	30:
		bBusy := TRUE;
		bPredictionPending := TRUE;
		IF fbMlSvr.Predict(
			pDataIn := ADR(stModelInput),
			nDataInSize := SIZEOF(ST_Wave41SmoothL1RobustLossInput),
			pDataOut := ADR(stModelOutput),
			nDataOutSize := SIZEOF(ST_Wave41SmoothL1RobustLossOutput),
			nTimeout := nPredictTimeout,
			nPriority := nPriority) THEN
			nErrorCode := fbMlSvr.nErrorCode;
			bError := fbMlSvr.bError OR (nErrorCode <> 0);
			nMaxInferenceDuration := fbMlSvr.nMaxInferenceDuration;
			bPredictionPending := FALSE;
			bBusy := FALSE;
			IF NOT(bError) THEN
				aPredictionOutput[0] := stModelOutput.out_prediction_tensor[0,0];
				FOR nOutputIndex := 1 TO 8 DO
					aPredictionOutput[nOutputIndex] := 0.0;
				END_FOR
				bPredictionReady := TRUE;
				nState := 20;
			ELSE
				nState := 90;
			END_IF
		END_IF

	90:
		bBusy := FALSE;
		bPredictionPending := FALSE;
		bError := TRUE;
END_CASE

nErrorCode := fbMlSvr.nErrorCode;
nMaxInferenceDuration := fbMlSvr.nMaxInferenceDuration;

END_FUNCTION_BLOCK

// ---- POUs/FB_Wave42GaussianNllTf3820Runner.TcPOU
FUNCTION_BLOCK FB_Wave42GaussianNllTf3820Runner
VAR_INPUT
	sModelJsonFilePath	: T_MaxString;
	sMlSvrNetId			: T_MaxString := 'local';
	eExecutionProvider	: E_ExecutionProvider := E_ExecutionProvider.CPU;
	bEnable				: BOOL;
	bReset					: BOOL;
	bLoadModel			: BOOL;
	nConfigureTimeout	: UDINT := 1000;
	nPredictTimeout		: UDINT := 100;
	nPriority			: UDINT := 0;
	fTheta					: REAL;
	fThetaDot				: REAL;
	fTorque				: REAL;
	fTemperature			: REAL;
	fDirectionFlag		: REAL;
	fThetaStep			: REAL := 0.25;
END_VAR
VAR
	fbMlSvr				: FB_MlSvrPrediction;
	stModelInput		: ST_Wave42GaussianNllInput;
	stModelOutput		: ST_Wave42GaussianNllOutput;
	rtrig_model			: R_TRIG;
	nState					: INT := 0;
	nSequenceIndex		: INT;
	nOutputIndex		: INT;
END_VAR
VAR_OUTPUT
	bConfigured			: BOOL;
	bBusy					: BOOL;
	bPredictionPending	: BOOL;
	bPredictionReady	: BOOL;
	bResetDone			: BOOL;
	bError					: BOOL;
	nErrorCode			: HRESULT;
	nMaxInferenceDuration	: UDINT;
	aPredictionOutput	: ARRAY[0..8] OF REAL;
END_VAR

rtrig_model(CLK := bLoadModel);

IF rtrig_model.Q THEN
	bPredictionPending := FALSE;
	bPredictionReady := FALSE;
	bResetDone := FALSE;
	bError := FALSE;
	IF fbMlSvr.bConfigured THEN
		nState := 5;
	ELSE
		bConfigured := FALSE;
		nState := 10;
	END_IF
END_IF

IF bReset THEN
	bPredictionPending := FALSE;
	bPredictionReady := FALSE;
	bError := FALSE;
	IF fbMlSvr.bConfigured THEN
		nState := 5;
	ELSE
		bConfigured := FALSE;
		bResetDone := TRUE;
		nState := 0;
	END_IF
END_IF

CASE nState OF
	0:
		bBusy := FALSE;
		IF bLoadModel AND NOT(bConfigured) AND NOT(bReset) THEN
			nState := 10;
		END_IF

	5:
		bBusy := TRUE;
		IF fbMlSvr.Deconfigure(nTimeout := nConfigureTimeout) THEN
			nErrorCode := fbMlSvr.nErrorCode;
			bError := fbMlSvr.bError OR (nErrorCode <> 0);
			bConfigured := FALSE;
			bBusy := FALSE;
			bResetDone := NOT(bError);
			IF bError THEN
				nState := 90;
			ELSIF bReset THEN
				nState := 0;
			ELSE
				nState := 10;
			END_IF
		END_IF

	10:
		bBusy := TRUE;
		fbMlSvr.stPredictionParameter.sMlModelFilePath := sModelJsonFilePath;
		fbMlSvr.stPredictionParameter.sMlSvrNetId := sMlSvrNetId;
		fbMlSvr.stPredictionParameter.eExecutionProvider := eExecutionProvider;
		IF fbMlSvr.Configure(nTimeout := nConfigureTimeout, nPriority := nPriority) THEN
			nErrorCode := fbMlSvr.nErrorCode;
			bError := fbMlSvr.bError OR (nErrorCode <> 0);
			bConfigured := fbMlSvr.bConfigured AND NOT(bError);
			bBusy := FALSE;
			IF bConfigured THEN
				nState := 20;
			ELSE
				nState := 90;
			END_IF
		END_IF

	20:
		bBusy := FALSE;
		bPredictionPending := FALSE;
		IF bEnable AND bConfigured AND NOT(bError) AND NOT(bReset) THEN
			FOR nSequenceIndex := 0 TO 32 DO
				stModelInput.in_input_tensor[0,nSequenceIndex,0] := fTheta + (INT_TO_REAL(nSequenceIndex) * fThetaStep);
				stModelInput.in_input_tensor[0,nSequenceIndex,1] := fThetaDot;
				stModelInput.in_input_tensor[0,nSequenceIndex,2] := fTorque;
				stModelInput.in_input_tensor[0,nSequenceIndex,3] := fTemperature;
			END_FOR
			bPredictionReady := FALSE;
			bPredictionPending := TRUE;
			nState := 30;
		END_IF

	30:
		bBusy := TRUE;
		bPredictionPending := TRUE;
		IF fbMlSvr.Predict(
			pDataIn := ADR(stModelInput),
			nDataInSize := SIZEOF(ST_Wave42GaussianNllInput),
			pDataOut := ADR(stModelOutput),
			nDataOutSize := SIZEOF(ST_Wave42GaussianNllOutput),
			nTimeout := nPredictTimeout,
			nPriority := nPriority) THEN
			nErrorCode := fbMlSvr.nErrorCode;
			bError := fbMlSvr.bError OR (nErrorCode <> 0);
			nMaxInferenceDuration := fbMlSvr.nMaxInferenceDuration;
			bPredictionPending := FALSE;
			bBusy := FALSE;
			IF NOT(bError) THEN
				aPredictionOutput[0] := stModelOutput.out_prediction_tensor[0,0];
				aPredictionOutput[1] := stModelOutput.out_prediction_tensor[0,1];
				FOR nOutputIndex := 2 TO 8 DO
					aPredictionOutput[nOutputIndex] := 0.0;
				END_FOR
				bPredictionReady := TRUE;
				nState := 20;
			ELSE
				nState := 90;
			END_IF
		END_IF

	90:
		bBusy := FALSE;
		bPredictionPending := FALSE;
		bError := TRUE;
END_CASE

nErrorCode := fbMlSvr.nErrorCode;
nMaxInferenceDuration := fbMlSvr.nMaxInferenceDuration;

END_FUNCTION_BLOCK

// ---- POUs/FB_Wave42QuantileP10P50P90Tf3820Runner.TcPOU
FUNCTION_BLOCK FB_Wave42QuantileP10P50P90Tf3820Runner
VAR_INPUT
	sModelJsonFilePath	: T_MaxString;
	sMlSvrNetId			: T_MaxString := 'local';
	eExecutionProvider	: E_ExecutionProvider := E_ExecutionProvider.CPU;
	bEnable				: BOOL;
	bReset					: BOOL;
	bLoadModel			: BOOL;
	nConfigureTimeout	: UDINT := 1000;
	nPredictTimeout		: UDINT := 100;
	nPriority			: UDINT := 0;
	fTheta					: REAL;
	fThetaDot				: REAL;
	fTorque				: REAL;
	fTemperature			: REAL;
	fDirectionFlag		: REAL;
	fThetaStep			: REAL := 0.25;
END_VAR
VAR
	fbMlSvr				: FB_MlSvrPrediction;
	stModelInput		: ST_Wave42QuantileP10P50P90Input;
	stModelOutput		: ST_Wave42QuantileP10P50P90Output;
	rtrig_model			: R_TRIG;
	nState					: INT := 0;
	nSequenceIndex		: INT;
	nOutputIndex		: INT;
END_VAR
VAR_OUTPUT
	bConfigured			: BOOL;
	bBusy					: BOOL;
	bPredictionPending	: BOOL;
	bPredictionReady	: BOOL;
	bResetDone			: BOOL;
	bError					: BOOL;
	nErrorCode			: HRESULT;
	nMaxInferenceDuration	: UDINT;
	aPredictionOutput	: ARRAY[0..8] OF REAL;
END_VAR

rtrig_model(CLK := bLoadModel);

IF rtrig_model.Q THEN
	bPredictionPending := FALSE;
	bPredictionReady := FALSE;
	bResetDone := FALSE;
	bError := FALSE;
	IF fbMlSvr.bConfigured THEN
		nState := 5;
	ELSE
		bConfigured := FALSE;
		nState := 10;
	END_IF
END_IF

IF bReset THEN
	bPredictionPending := FALSE;
	bPredictionReady := FALSE;
	bError := FALSE;
	IF fbMlSvr.bConfigured THEN
		nState := 5;
	ELSE
		bConfigured := FALSE;
		bResetDone := TRUE;
		nState := 0;
	END_IF
END_IF

CASE nState OF
	0:
		bBusy := FALSE;
		IF bLoadModel AND NOT(bConfigured) AND NOT(bReset) THEN
			nState := 10;
		END_IF

	5:
		bBusy := TRUE;
		IF fbMlSvr.Deconfigure(nTimeout := nConfigureTimeout) THEN
			nErrorCode := fbMlSvr.nErrorCode;
			bError := fbMlSvr.bError OR (nErrorCode <> 0);
			bConfigured := FALSE;
			bBusy := FALSE;
			bResetDone := NOT(bError);
			IF bError THEN
				nState := 90;
			ELSIF bReset THEN
				nState := 0;
			ELSE
				nState := 10;
			END_IF
		END_IF

	10:
		bBusy := TRUE;
		fbMlSvr.stPredictionParameter.sMlModelFilePath := sModelJsonFilePath;
		fbMlSvr.stPredictionParameter.sMlSvrNetId := sMlSvrNetId;
		fbMlSvr.stPredictionParameter.eExecutionProvider := eExecutionProvider;
		IF fbMlSvr.Configure(nTimeout := nConfigureTimeout, nPriority := nPriority) THEN
			nErrorCode := fbMlSvr.nErrorCode;
			bError := fbMlSvr.bError OR (nErrorCode <> 0);
			bConfigured := fbMlSvr.bConfigured AND NOT(bError);
			bBusy := FALSE;
			IF bConfigured THEN
				nState := 20;
			ELSE
				nState := 90;
			END_IF
		END_IF

	20:
		bBusy := FALSE;
		bPredictionPending := FALSE;
		IF bEnable AND bConfigured AND NOT(bError) AND NOT(bReset) THEN
			FOR nSequenceIndex := 0 TO 32 DO
				stModelInput.in_input_tensor[0,nSequenceIndex,0] := fTheta + (INT_TO_REAL(nSequenceIndex) * fThetaStep);
				stModelInput.in_input_tensor[0,nSequenceIndex,1] := fThetaDot;
				stModelInput.in_input_tensor[0,nSequenceIndex,2] := fTorque;
				stModelInput.in_input_tensor[0,nSequenceIndex,3] := fTemperature;
			END_FOR
			bPredictionReady := FALSE;
			bPredictionPending := TRUE;
			nState := 30;
		END_IF

	30:
		bBusy := TRUE;
		bPredictionPending := TRUE;
		IF fbMlSvr.Predict(
			pDataIn := ADR(stModelInput),
			nDataInSize := SIZEOF(ST_Wave42QuantileP10P50P90Input),
			pDataOut := ADR(stModelOutput),
			nDataOutSize := SIZEOF(ST_Wave42QuantileP10P50P90Output),
			nTimeout := nPredictTimeout,
			nPriority := nPriority) THEN
			nErrorCode := fbMlSvr.nErrorCode;
			bError := fbMlSvr.bError OR (nErrorCode <> 0);
			nMaxInferenceDuration := fbMlSvr.nMaxInferenceDuration;
			bPredictionPending := FALSE;
			bBusy := FALSE;
			IF NOT(bError) THEN
				aPredictionOutput[0] := stModelOutput.out_prediction_tensor[0,0];
				aPredictionOutput[1] := stModelOutput.out_prediction_tensor[0,1];
				aPredictionOutput[2] := stModelOutput.out_prediction_tensor[0,2];
				FOR nOutputIndex := 3 TO 8 DO
					aPredictionOutput[nOutputIndex] := 0.0;
				END_FOR
				bPredictionReady := TRUE;
				nState := 20;
			ELSE
				nState := 90;
			END_IF
		END_IF

	90:
		bBusy := FALSE;
		bPredictionPending := FALSE;
		bError := TRUE;
END_CASE

nErrorCode := fbMlSvr.nErrorCode;
nMaxInferenceDuration := fbMlSvr.nMaxInferenceDuration;

END_FUNCTION_BLOCK

// ---- POUs/FB_Wave43MixtureDensityK2Tf3820Runner.TcPOU
FUNCTION_BLOCK FB_Wave43MixtureDensityK2Tf3820Runner
VAR_INPUT
	sModelJsonFilePath	: T_MaxString;
	sMlSvrNetId			: T_MaxString := 'local';
	eExecutionProvider	: E_ExecutionProvider := E_ExecutionProvider.CPU;
	bEnable				: BOOL;
	bReset					: BOOL;
	bLoadModel			: BOOL;
	nConfigureTimeout	: UDINT := 1000;
	nPredictTimeout		: UDINT := 100;
	nPriority			: UDINT := 0;
	fTheta					: REAL;
	fThetaDot				: REAL;
	fTorque				: REAL;
	fTemperature			: REAL;
	fDirectionFlag		: REAL;
	fThetaStep			: REAL := 0.25;
END_VAR
VAR
	fbMlSvr				: FB_MlSvrPrediction;
	stModelInput		: ST_Wave43MixtureDensityK2Input;
	stModelOutput		: ST_Wave43MixtureDensityK2Output;
	rtrig_model			: R_TRIG;
	nState					: INT := 0;
	nSequenceIndex		: INT;
	nOutputIndex		: INT;
END_VAR
VAR_OUTPUT
	bConfigured			: BOOL;
	bBusy					: BOOL;
	bPredictionPending	: BOOL;
	bPredictionReady	: BOOL;
	bResetDone			: BOOL;
	bError					: BOOL;
	nErrorCode			: HRESULT;
	nMaxInferenceDuration	: UDINT;
	aPredictionOutput	: ARRAY[0..8] OF REAL;
END_VAR

rtrig_model(CLK := bLoadModel);

IF rtrig_model.Q THEN
	bPredictionPending := FALSE;
	bPredictionReady := FALSE;
	bResetDone := FALSE;
	bError := FALSE;
	IF fbMlSvr.bConfigured THEN
		nState := 5;
	ELSE
		bConfigured := FALSE;
		nState := 10;
	END_IF
END_IF

IF bReset THEN
	bPredictionPending := FALSE;
	bPredictionReady := FALSE;
	bError := FALSE;
	IF fbMlSvr.bConfigured THEN
		nState := 5;
	ELSE
		bConfigured := FALSE;
		bResetDone := TRUE;
		nState := 0;
	END_IF
END_IF

CASE nState OF
	0:
		bBusy := FALSE;
		IF bLoadModel AND NOT(bConfigured) AND NOT(bReset) THEN
			nState := 10;
		END_IF

	5:
		bBusy := TRUE;
		IF fbMlSvr.Deconfigure(nTimeout := nConfigureTimeout) THEN
			nErrorCode := fbMlSvr.nErrorCode;
			bError := fbMlSvr.bError OR (nErrorCode <> 0);
			bConfigured := FALSE;
			bBusy := FALSE;
			bResetDone := NOT(bError);
			IF bError THEN
				nState := 90;
			ELSIF bReset THEN
				nState := 0;
			ELSE
				nState := 10;
			END_IF
		END_IF

	10:
		bBusy := TRUE;
		fbMlSvr.stPredictionParameter.sMlModelFilePath := sModelJsonFilePath;
		fbMlSvr.stPredictionParameter.sMlSvrNetId := sMlSvrNetId;
		fbMlSvr.stPredictionParameter.eExecutionProvider := eExecutionProvider;
		IF fbMlSvr.Configure(nTimeout := nConfigureTimeout, nPriority := nPriority) THEN
			nErrorCode := fbMlSvr.nErrorCode;
			bError := fbMlSvr.bError OR (nErrorCode <> 0);
			bConfigured := fbMlSvr.bConfigured AND NOT(bError);
			bBusy := FALSE;
			IF bConfigured THEN
				nState := 20;
			ELSE
				nState := 90;
			END_IF
		END_IF

	20:
		bBusy := FALSE;
		bPredictionPending := FALSE;
		IF bEnable AND bConfigured AND NOT(bError) AND NOT(bReset) THEN
			FOR nSequenceIndex := 0 TO 32 DO
				stModelInput.in_input_tensor[0,nSequenceIndex,0] := fTheta + (INT_TO_REAL(nSequenceIndex) * fThetaStep);
				stModelInput.in_input_tensor[0,nSequenceIndex,1] := fThetaDot;
				stModelInput.in_input_tensor[0,nSequenceIndex,2] := fTorque;
				stModelInput.in_input_tensor[0,nSequenceIndex,3] := fTemperature;
			END_FOR
			bPredictionReady := FALSE;
			bPredictionPending := TRUE;
			nState := 30;
		END_IF

	30:
		bBusy := TRUE;
		bPredictionPending := TRUE;
		IF fbMlSvr.Predict(
			pDataIn := ADR(stModelInput),
			nDataInSize := SIZEOF(ST_Wave43MixtureDensityK2Input),
			pDataOut := ADR(stModelOutput),
			nDataOutSize := SIZEOF(ST_Wave43MixtureDensityK2Output),
			nTimeout := nPredictTimeout,
			nPriority := nPriority) THEN
			nErrorCode := fbMlSvr.nErrorCode;
			bError := fbMlSvr.bError OR (nErrorCode <> 0);
			nMaxInferenceDuration := fbMlSvr.nMaxInferenceDuration;
			bPredictionPending := FALSE;
			bBusy := FALSE;
			IF NOT(bError) THEN
				aPredictionOutput[0] := stModelOutput.out_prediction_tensor[0,0];
				aPredictionOutput[1] := stModelOutput.out_prediction_tensor[0,1];
				aPredictionOutput[2] := stModelOutput.out_prediction_tensor[0,2];
				aPredictionOutput[3] := stModelOutput.out_prediction_tensor[0,3];
				aPredictionOutput[4] := stModelOutput.out_prediction_tensor[0,4];
				aPredictionOutput[5] := stModelOutput.out_prediction_tensor[0,5];
				FOR nOutputIndex := 6 TO 8 DO
					aPredictionOutput[nOutputIndex] := 0.0;
				END_FOR
				bPredictionReady := TRUE;
				nState := 20;
			ELSE
				nState := 90;
			END_IF
		END_IF

	90:
		bBusy := FALSE;
		bPredictionPending := FALSE;
		bError := TRUE;
END_CASE

nErrorCode := fbMlSvr.nErrorCode;
nMaxInferenceDuration := fbMlSvr.nMaxInferenceDuration;

END_FUNCTION_BLOCK

// ---- POUs/FB_Wave43MixtureDensityK3Tf3820Runner.TcPOU
FUNCTION_BLOCK FB_Wave43MixtureDensityK3Tf3820Runner
VAR_INPUT
	sModelJsonFilePath	: T_MaxString;
	sMlSvrNetId			: T_MaxString := 'local';
	eExecutionProvider	: E_ExecutionProvider := E_ExecutionProvider.CPU;
	bEnable				: BOOL;
	bReset					: BOOL;
	bLoadModel			: BOOL;
	nConfigureTimeout	: UDINT := 1000;
	nPredictTimeout		: UDINT := 100;
	nPriority			: UDINT := 0;
	fTheta					: REAL;
	fThetaDot				: REAL;
	fTorque				: REAL;
	fTemperature			: REAL;
	fDirectionFlag		: REAL;
	fThetaStep			: REAL := 0.25;
END_VAR
VAR
	fbMlSvr				: FB_MlSvrPrediction;
	stModelInput		: ST_Wave43MixtureDensityK3Input;
	stModelOutput		: ST_Wave43MixtureDensityK3Output;
	rtrig_model			: R_TRIG;
	nState					: INT := 0;
	nSequenceIndex		: INT;
	nOutputIndex		: INT;
END_VAR
VAR_OUTPUT
	bConfigured			: BOOL;
	bBusy					: BOOL;
	bPredictionPending	: BOOL;
	bPredictionReady	: BOOL;
	bResetDone			: BOOL;
	bError					: BOOL;
	nErrorCode			: HRESULT;
	nMaxInferenceDuration	: UDINT;
	aPredictionOutput	: ARRAY[0..8] OF REAL;
END_VAR

rtrig_model(CLK := bLoadModel);

IF rtrig_model.Q THEN
	bPredictionPending := FALSE;
	bPredictionReady := FALSE;
	bResetDone := FALSE;
	bError := FALSE;
	IF fbMlSvr.bConfigured THEN
		nState := 5;
	ELSE
		bConfigured := FALSE;
		nState := 10;
	END_IF
END_IF

IF bReset THEN
	bPredictionPending := FALSE;
	bPredictionReady := FALSE;
	bError := FALSE;
	IF fbMlSvr.bConfigured THEN
		nState := 5;
	ELSE
		bConfigured := FALSE;
		bResetDone := TRUE;
		nState := 0;
	END_IF
END_IF

CASE nState OF
	0:
		bBusy := FALSE;
		IF bLoadModel AND NOT(bConfigured) AND NOT(bReset) THEN
			nState := 10;
		END_IF

	5:
		bBusy := TRUE;
		IF fbMlSvr.Deconfigure(nTimeout := nConfigureTimeout) THEN
			nErrorCode := fbMlSvr.nErrorCode;
			bError := fbMlSvr.bError OR (nErrorCode <> 0);
			bConfigured := FALSE;
			bBusy := FALSE;
			bResetDone := NOT(bError);
			IF bError THEN
				nState := 90;
			ELSIF bReset THEN
				nState := 0;
			ELSE
				nState := 10;
			END_IF
		END_IF

	10:
		bBusy := TRUE;
		fbMlSvr.stPredictionParameter.sMlModelFilePath := sModelJsonFilePath;
		fbMlSvr.stPredictionParameter.sMlSvrNetId := sMlSvrNetId;
		fbMlSvr.stPredictionParameter.eExecutionProvider := eExecutionProvider;
		IF fbMlSvr.Configure(nTimeout := nConfigureTimeout, nPriority := nPriority) THEN
			nErrorCode := fbMlSvr.nErrorCode;
			bError := fbMlSvr.bError OR (nErrorCode <> 0);
			bConfigured := fbMlSvr.bConfigured AND NOT(bError);
			bBusy := FALSE;
			IF bConfigured THEN
				nState := 20;
			ELSE
				nState := 90;
			END_IF
		END_IF

	20:
		bBusy := FALSE;
		bPredictionPending := FALSE;
		IF bEnable AND bConfigured AND NOT(bError) AND NOT(bReset) THEN
			FOR nSequenceIndex := 0 TO 32 DO
				stModelInput.in_input_tensor[0,nSequenceIndex,0] := fTheta + (INT_TO_REAL(nSequenceIndex) * fThetaStep);
				stModelInput.in_input_tensor[0,nSequenceIndex,1] := fThetaDot;
				stModelInput.in_input_tensor[0,nSequenceIndex,2] := fTorque;
				stModelInput.in_input_tensor[0,nSequenceIndex,3] := fTemperature;
			END_FOR
			bPredictionReady := FALSE;
			bPredictionPending := TRUE;
			nState := 30;
		END_IF

	30:
		bBusy := TRUE;
		bPredictionPending := TRUE;
		IF fbMlSvr.Predict(
			pDataIn := ADR(stModelInput),
			nDataInSize := SIZEOF(ST_Wave43MixtureDensityK3Input),
			pDataOut := ADR(stModelOutput),
			nDataOutSize := SIZEOF(ST_Wave43MixtureDensityK3Output),
			nTimeout := nPredictTimeout,
			nPriority := nPriority) THEN
			nErrorCode := fbMlSvr.nErrorCode;
			bError := fbMlSvr.bError OR (nErrorCode <> 0);
			nMaxInferenceDuration := fbMlSvr.nMaxInferenceDuration;
			bPredictionPending := FALSE;
			bBusy := FALSE;
			IF NOT(bError) THEN
				aPredictionOutput[0] := stModelOutput.out_prediction_tensor[0,0];
				aPredictionOutput[1] := stModelOutput.out_prediction_tensor[0,1];
				aPredictionOutput[2] := stModelOutput.out_prediction_tensor[0,2];
				aPredictionOutput[3] := stModelOutput.out_prediction_tensor[0,3];
				aPredictionOutput[4] := stModelOutput.out_prediction_tensor[0,4];
				aPredictionOutput[5] := stModelOutput.out_prediction_tensor[0,5];
				aPredictionOutput[6] := stModelOutput.out_prediction_tensor[0,6];
				aPredictionOutput[7] := stModelOutput.out_prediction_tensor[0,7];
				aPredictionOutput[8] := stModelOutput.out_prediction_tensor[0,8];
				bPredictionReady := TRUE;
				nState := 20;
			ELSE
				nState := 90;
			END_IF
		END_IF

	90:
		bBusy := FALSE;
		bPredictionPending := FALSE;
		bError := TRUE;
END_CASE

nErrorCode := fbMlSvr.nErrorCode;
nMaxInferenceDuration := fbMlSvr.nMaxInferenceDuration;

END_FUNCTION_BLOCK

// ---- POUs/FB_Wave44CausalTcnLatentOffsetResidualTf3820Runner.TcPOU
FUNCTION_BLOCK FB_Wave44CausalTcnLatentOffsetResidualTf3820Runner
VAR_INPUT
	sModelJsonFilePath	: T_MaxString;
	sMlSvrNetId			: T_MaxString := 'local';
	eExecutionProvider	: E_ExecutionProvider := E_ExecutionProvider.CPU;
	bEnable				: BOOL;
	bReset					: BOOL;
	bLoadModel			: BOOL;
	nConfigureTimeout	: UDINT := 1000;
	nPredictTimeout		: UDINT := 100;
	nPriority			: UDINT := 0;
	fTheta					: REAL;
	fThetaDot				: REAL;
	fTorque				: REAL;
	fTemperature			: REAL;
	fDirectionFlag		: REAL;
	fThetaStep			: REAL := 0.25;
END_VAR
VAR
	fbMlSvr				: FB_MlSvrPrediction;
	stModelInput		: ST_Wave44CausalTcnLatentOffsetResidualInput;
	stModelOutput		: ST_Wave44CausalTcnLatentOffsetResidualOutput;
	rtrig_model			: R_TRIG;
	nState					: INT := 0;
	nSequenceIndex		: INT;
	nOutputIndex		: INT;
END_VAR
VAR_OUTPUT
	bConfigured			: BOOL;
	bBusy					: BOOL;
	bPredictionPending	: BOOL;
	bPredictionReady	: BOOL;
	bResetDone			: BOOL;
	bError					: BOOL;
	nErrorCode			: HRESULT;
	nMaxInferenceDuration	: UDINT;
	aPredictionOutput	: ARRAY[0..8] OF REAL;
END_VAR

rtrig_model(CLK := bLoadModel);

IF rtrig_model.Q THEN
	bPredictionPending := FALSE;
	bPredictionReady := FALSE;
	bResetDone := FALSE;
	bError := FALSE;
	IF fbMlSvr.bConfigured THEN
		nState := 5;
	ELSE
		bConfigured := FALSE;
		nState := 10;
	END_IF
END_IF

IF bReset THEN
	bPredictionPending := FALSE;
	bPredictionReady := FALSE;
	bError := FALSE;
	IF fbMlSvr.bConfigured THEN
		nState := 5;
	ELSE
		bConfigured := FALSE;
		bResetDone := TRUE;
		nState := 0;
	END_IF
END_IF

CASE nState OF
	0:
		bBusy := FALSE;
		IF bLoadModel AND NOT(bConfigured) AND NOT(bReset) THEN
			nState := 10;
		END_IF

	5:
		bBusy := TRUE;
		IF fbMlSvr.Deconfigure(nTimeout := nConfigureTimeout) THEN
			nErrorCode := fbMlSvr.nErrorCode;
			bError := fbMlSvr.bError OR (nErrorCode <> 0);
			bConfigured := FALSE;
			bBusy := FALSE;
			bResetDone := NOT(bError);
			IF bError THEN
				nState := 90;
			ELSIF bReset THEN
				nState := 0;
			ELSE
				nState := 10;
			END_IF
		END_IF

	10:
		bBusy := TRUE;
		fbMlSvr.stPredictionParameter.sMlModelFilePath := sModelJsonFilePath;
		fbMlSvr.stPredictionParameter.sMlSvrNetId := sMlSvrNetId;
		fbMlSvr.stPredictionParameter.eExecutionProvider := eExecutionProvider;
		IF fbMlSvr.Configure(nTimeout := nConfigureTimeout, nPriority := nPriority) THEN
			nErrorCode := fbMlSvr.nErrorCode;
			bError := fbMlSvr.bError OR (nErrorCode <> 0);
			bConfigured := fbMlSvr.bConfigured AND NOT(bError);
			bBusy := FALSE;
			IF bConfigured THEN
				nState := 20;
			ELSE
				nState := 90;
			END_IF
		END_IF

	20:
		bBusy := FALSE;
		bPredictionPending := FALSE;
		IF bEnable AND bConfigured AND NOT(bError) AND NOT(bReset) THEN
			FOR nSequenceIndex := 0 TO 32 DO
				stModelInput.in_input_tensor[0,nSequenceIndex,0] := fTheta + (INT_TO_REAL(nSequenceIndex) * fThetaStep);
				stModelInput.in_input_tensor[0,nSequenceIndex,1] := fThetaDot;
				stModelInput.in_input_tensor[0,nSequenceIndex,2] := fTorque;
				stModelInput.in_input_tensor[0,nSequenceIndex,3] := fTemperature;
			END_FOR
			bPredictionReady := FALSE;
			bPredictionPending := TRUE;
			nState := 30;
		END_IF

	30:
		bBusy := TRUE;
		bPredictionPending := TRUE;
		IF fbMlSvr.Predict(
			pDataIn := ADR(stModelInput),
			nDataInSize := SIZEOF(ST_Wave44CausalTcnLatentOffsetResidualInput),
			pDataOut := ADR(stModelOutput),
			nDataOutSize := SIZEOF(ST_Wave44CausalTcnLatentOffsetResidualOutput),
			nTimeout := nPredictTimeout,
			nPriority := nPriority) THEN
			nErrorCode := fbMlSvr.nErrorCode;
			bError := fbMlSvr.bError OR (nErrorCode <> 0);
			nMaxInferenceDuration := fbMlSvr.nMaxInferenceDuration;
			bPredictionPending := FALSE;
			bBusy := FALSE;
			IF NOT(bError) THEN
				aPredictionOutput[0] := stModelOutput.out_prediction_tensor[0,0];
				FOR nOutputIndex := 1 TO 8 DO
					aPredictionOutput[nOutputIndex] := 0.0;
				END_FOR
				bPredictionReady := TRUE;
				nState := 20;
			ELSE
				nState := 90;
			END_IF
		END_IF

	90:
		bBusy := FALSE;
		bPredictionPending := FALSE;
		bError := TRUE;
END_CASE

nErrorCode := fbMlSvr.nErrorCode;
nMaxInferenceDuration := fbMlSvr.nMaxInferenceDuration;

END_FUNCTION_BLOCK

// ---- POUs/FB_Wave44GruLatentOffsetResidualTf3820Runner.TcPOU
FUNCTION_BLOCK FB_Wave44GruLatentOffsetResidualTf3820Runner
VAR_INPUT
	sModelJsonFilePath	: T_MaxString;
	sMlSvrNetId			: T_MaxString := 'local';
	eExecutionProvider	: E_ExecutionProvider := E_ExecutionProvider.CPU;
	bEnable				: BOOL;
	bReset					: BOOL;
	bLoadModel			: BOOL;
	nConfigureTimeout	: UDINT := 1000;
	nPredictTimeout		: UDINT := 100;
	nPriority			: UDINT := 0;
	fTheta					: REAL;
	fThetaDot				: REAL;
	fTorque				: REAL;
	fTemperature			: REAL;
	fDirectionFlag		: REAL;
	fThetaStep			: REAL := 0.25;
END_VAR
VAR
	fbMlSvr				: FB_MlSvrPrediction;
	stModelInput		: ST_Wave44GruLatentOffsetResidualInput;
	stModelOutput		: ST_Wave44GruLatentOffsetResidualOutput;
	rtrig_model			: R_TRIG;
	nState					: INT := 0;
	nSequenceIndex		: INT;
	nOutputIndex		: INT;
END_VAR
VAR_OUTPUT
	bConfigured			: BOOL;
	bBusy					: BOOL;
	bPredictionPending	: BOOL;
	bPredictionReady	: BOOL;
	bResetDone			: BOOL;
	bError					: BOOL;
	nErrorCode			: HRESULT;
	nMaxInferenceDuration	: UDINT;
	aPredictionOutput	: ARRAY[0..8] OF REAL;
END_VAR

rtrig_model(CLK := bLoadModel);

IF rtrig_model.Q THEN
	bPredictionPending := FALSE;
	bPredictionReady := FALSE;
	bResetDone := FALSE;
	bError := FALSE;
	IF fbMlSvr.bConfigured THEN
		nState := 5;
	ELSE
		bConfigured := FALSE;
		nState := 10;
	END_IF
END_IF

IF bReset THEN
	bPredictionPending := FALSE;
	bPredictionReady := FALSE;
	bError := FALSE;
	IF fbMlSvr.bConfigured THEN
		nState := 5;
	ELSE
		bConfigured := FALSE;
		bResetDone := TRUE;
		nState := 0;
	END_IF
END_IF

CASE nState OF
	0:
		bBusy := FALSE;
		IF bLoadModel AND NOT(bConfigured) AND NOT(bReset) THEN
			nState := 10;
		END_IF

	5:
		bBusy := TRUE;
		IF fbMlSvr.Deconfigure(nTimeout := nConfigureTimeout) THEN
			nErrorCode := fbMlSvr.nErrorCode;
			bError := fbMlSvr.bError OR (nErrorCode <> 0);
			bConfigured := FALSE;
			bBusy := FALSE;
			bResetDone := NOT(bError);
			IF bError THEN
				nState := 90;
			ELSIF bReset THEN
				nState := 0;
			ELSE
				nState := 10;
			END_IF
		END_IF

	10:
		bBusy := TRUE;
		fbMlSvr.stPredictionParameter.sMlModelFilePath := sModelJsonFilePath;
		fbMlSvr.stPredictionParameter.sMlSvrNetId := sMlSvrNetId;
		fbMlSvr.stPredictionParameter.eExecutionProvider := eExecutionProvider;
		IF fbMlSvr.Configure(nTimeout := nConfigureTimeout, nPriority := nPriority) THEN
			nErrorCode := fbMlSvr.nErrorCode;
			bError := fbMlSvr.bError OR (nErrorCode <> 0);
			bConfigured := fbMlSvr.bConfigured AND NOT(bError);
			bBusy := FALSE;
			IF bConfigured THEN
				nState := 20;
			ELSE
				nState := 90;
			END_IF
		END_IF

	20:
		bBusy := FALSE;
		bPredictionPending := FALSE;
		IF bEnable AND bConfigured AND NOT(bError) AND NOT(bReset) THEN
			FOR nSequenceIndex := 0 TO 32 DO
				stModelInput.in_input_tensor[0,nSequenceIndex,0] := fTheta + (INT_TO_REAL(nSequenceIndex) * fThetaStep);
				stModelInput.in_input_tensor[0,nSequenceIndex,1] := fThetaDot;
				stModelInput.in_input_tensor[0,nSequenceIndex,2] := fTorque;
				stModelInput.in_input_tensor[0,nSequenceIndex,3] := fTemperature;
			END_FOR
			bPredictionReady := FALSE;
			bPredictionPending := TRUE;
			nState := 30;
		END_IF

	30:
		bBusy := TRUE;
		bPredictionPending := TRUE;
		IF fbMlSvr.Predict(
			pDataIn := ADR(stModelInput),
			nDataInSize := SIZEOF(ST_Wave44GruLatentOffsetResidualInput),
			pDataOut := ADR(stModelOutput),
			nDataOutSize := SIZEOF(ST_Wave44GruLatentOffsetResidualOutput),
			nTimeout := nPredictTimeout,
			nPriority := nPriority) THEN
			nErrorCode := fbMlSvr.nErrorCode;
			bError := fbMlSvr.bError OR (nErrorCode <> 0);
			nMaxInferenceDuration := fbMlSvr.nMaxInferenceDuration;
			bPredictionPending := FALSE;
			bBusy := FALSE;
			IF NOT(bError) THEN
				aPredictionOutput[0] := stModelOutput.out_prediction_tensor[0,0];
				FOR nOutputIndex := 1 TO 8 DO
					aPredictionOutput[nOutputIndex] := 0.0;
				END_FOR
				bPredictionReady := TRUE;
				nState := 20;
			ELSE
				nState := 90;
			END_IF
		END_IF

	90:
		bBusy := FALSE;
		bPredictionPending := FALSE;
		bError := TRUE;
END_CASE

nErrorCode := fbMlSvr.nErrorCode;
nMaxInferenceDuration := fbMlSvr.nMaxInferenceDuration;

END_FUNCTION_BLOCK

// ---- POUs/FB_Wave51HarmonicPriorPointwiseControlTf3820Runner.TcPOU
FUNCTION_BLOCK FB_Wave51HarmonicPriorPointwiseControlTf3820Runner
VAR_INPUT
	sModelJsonFilePath	: T_MaxString;
	sMlSvrNetId			: T_MaxString := 'local';
	eExecutionProvider	: E_ExecutionProvider := E_ExecutionProvider.CPU;
	bEnable				: BOOL;
	bReset					: BOOL;
	bLoadModel			: BOOL;
	nConfigureTimeout	: UDINT := 1000;
	nPredictTimeout		: UDINT := 100;
	nPriority			: UDINT := 0;
	fTheta					: REAL;
	fThetaDot				: REAL;
	fTorque				: REAL;
	fTemperature			: REAL;
	fDirectionFlag		: REAL;
	fThetaStep			: REAL := 0.25;
END_VAR
VAR
	fbMlSvr				: FB_MlSvrPrediction;
	stModelInput		: ST_Wave51HarmonicPriorPointwiseControlInput;
	stModelOutput		: ST_Wave51HarmonicPriorPointwiseControlOutput;
	rtrig_model			: R_TRIG;
	nState					: INT := 0;
	nSequenceIndex		: INT;
	nOutputIndex		: INT;
END_VAR
VAR_OUTPUT
	bConfigured			: BOOL;
	bBusy					: BOOL;
	bPredictionPending	: BOOL;
	bPredictionReady	: BOOL;
	bResetDone			: BOOL;
	bError					: BOOL;
	nErrorCode			: HRESULT;
	nMaxInferenceDuration	: UDINT;
	aPredictionOutput	: ARRAY[0..8] OF REAL;
END_VAR

rtrig_model(CLK := bLoadModel);

IF rtrig_model.Q THEN
	bPredictionPending := FALSE;
	bPredictionReady := FALSE;
	bResetDone := FALSE;
	bError := FALSE;
	IF fbMlSvr.bConfigured THEN
		nState := 5;
	ELSE
		bConfigured := FALSE;
		nState := 10;
	END_IF
END_IF

IF bReset THEN
	bPredictionPending := FALSE;
	bPredictionReady := FALSE;
	bError := FALSE;
	IF fbMlSvr.bConfigured THEN
		nState := 5;
	ELSE
		bConfigured := FALSE;
		bResetDone := TRUE;
		nState := 0;
	END_IF
END_IF

CASE nState OF
	0:
		bBusy := FALSE;
		IF bLoadModel AND NOT(bConfigured) AND NOT(bReset) THEN
			nState := 10;
		END_IF

	5:
		bBusy := TRUE;
		IF fbMlSvr.Deconfigure(nTimeout := nConfigureTimeout) THEN
			nErrorCode := fbMlSvr.nErrorCode;
			bError := fbMlSvr.bError OR (nErrorCode <> 0);
			bConfigured := FALSE;
			bBusy := FALSE;
			bResetDone := NOT(bError);
			IF bError THEN
				nState := 90;
			ELSIF bReset THEN
				nState := 0;
			ELSE
				nState := 10;
			END_IF
		END_IF

	10:
		bBusy := TRUE;
		fbMlSvr.stPredictionParameter.sMlModelFilePath := sModelJsonFilePath;
		fbMlSvr.stPredictionParameter.sMlSvrNetId := sMlSvrNetId;
		fbMlSvr.stPredictionParameter.eExecutionProvider := eExecutionProvider;
		IF fbMlSvr.Configure(nTimeout := nConfigureTimeout, nPriority := nPriority) THEN
			nErrorCode := fbMlSvr.nErrorCode;
			bError := fbMlSvr.bError OR (nErrorCode <> 0);
			bConfigured := fbMlSvr.bConfigured AND NOT(bError);
			bBusy := FALSE;
			IF bConfigured THEN
				nState := 20;
			ELSE
				nState := 90;
			END_IF
		END_IF

	20:
		bBusy := FALSE;
		bPredictionPending := FALSE;
		IF bEnable AND bConfigured AND NOT(bError) AND NOT(bReset) THEN
			FOR nSequenceIndex := 0 TO 32 DO
				stModelInput.in_input_tensor[0,nSequenceIndex,0] := fTheta + (INT_TO_REAL(nSequenceIndex) * fThetaStep);
				stModelInput.in_input_tensor[0,nSequenceIndex,1] := fThetaDot;
				stModelInput.in_input_tensor[0,nSequenceIndex,2] := fTorque;
				stModelInput.in_input_tensor[0,nSequenceIndex,3] := fTemperature;
			END_FOR
			bPredictionReady := FALSE;
			bPredictionPending := TRUE;
			nState := 30;
		END_IF

	30:
		bBusy := TRUE;
		bPredictionPending := TRUE;
		IF fbMlSvr.Predict(
			pDataIn := ADR(stModelInput),
			nDataInSize := SIZEOF(ST_Wave51HarmonicPriorPointwiseControlInput),
			pDataOut := ADR(stModelOutput),
			nDataOutSize := SIZEOF(ST_Wave51HarmonicPriorPointwiseControlOutput),
			nTimeout := nPredictTimeout,
			nPriority := nPriority) THEN
			nErrorCode := fbMlSvr.nErrorCode;
			bError := fbMlSvr.bError OR (nErrorCode <> 0);
			nMaxInferenceDuration := fbMlSvr.nMaxInferenceDuration;
			bPredictionPending := FALSE;
			bBusy := FALSE;
			IF NOT(bError) THEN
				aPredictionOutput[0] := stModelOutput.out_prediction_tensor[0,0];
				FOR nOutputIndex := 1 TO 8 DO
					aPredictionOutput[nOutputIndex] := 0.0;
				END_FOR
				bPredictionReady := TRUE;
				nState := 20;
			ELSE
				nState := 90;
			END_IF
		END_IF

	90:
		bBusy := FALSE;
		bPredictionPending := FALSE;
		bError := TRUE;
END_CASE

nErrorCode := fbMlSvr.nErrorCode;
nMaxInferenceDuration := fbMlSvr.nMaxInferenceDuration;

END_FUNCTION_BLOCK

// ---- POUs/FB_Wave51HarmonicPriorSmoothL1StructuredTf3820Runner.TcPOU
FUNCTION_BLOCK FB_Wave51HarmonicPriorSmoothL1StructuredTf3820Runner
VAR_INPUT
	sModelJsonFilePath	: T_MaxString;
	sMlSvrNetId			: T_MaxString := 'local';
	eExecutionProvider	: E_ExecutionProvider := E_ExecutionProvider.CPU;
	bEnable				: BOOL;
	bReset					: BOOL;
	bLoadModel			: BOOL;
	nConfigureTimeout	: UDINT := 1000;
	nPredictTimeout		: UDINT := 100;
	nPriority			: UDINT := 0;
	fTheta					: REAL;
	fThetaDot				: REAL;
	fTorque				: REAL;
	fTemperature			: REAL;
	fDirectionFlag		: REAL;
	fThetaStep			: REAL := 0.25;
END_VAR
VAR
	fbMlSvr				: FB_MlSvrPrediction;
	stModelInput		: ST_Wave51HarmonicPriorSmoothL1StructuredInput;
	stModelOutput		: ST_Wave51HarmonicPriorSmoothL1StructuredOutput;
	rtrig_model			: R_TRIG;
	nState					: INT := 0;
	nSequenceIndex		: INT;
	nOutputIndex		: INT;
END_VAR
VAR_OUTPUT
	bConfigured			: BOOL;
	bBusy					: BOOL;
	bPredictionPending	: BOOL;
	bPredictionReady	: BOOL;
	bResetDone			: BOOL;
	bError					: BOOL;
	nErrorCode			: HRESULT;
	nMaxInferenceDuration	: UDINT;
	aPredictionOutput	: ARRAY[0..8] OF REAL;
END_VAR

rtrig_model(CLK := bLoadModel);

IF rtrig_model.Q THEN
	bPredictionPending := FALSE;
	bPredictionReady := FALSE;
	bResetDone := FALSE;
	bError := FALSE;
	IF fbMlSvr.bConfigured THEN
		nState := 5;
	ELSE
		bConfigured := FALSE;
		nState := 10;
	END_IF
END_IF

IF bReset THEN
	bPredictionPending := FALSE;
	bPredictionReady := FALSE;
	bError := FALSE;
	IF fbMlSvr.bConfigured THEN
		nState := 5;
	ELSE
		bConfigured := FALSE;
		bResetDone := TRUE;
		nState := 0;
	END_IF
END_IF

CASE nState OF
	0:
		bBusy := FALSE;
		IF bLoadModel AND NOT(bConfigured) AND NOT(bReset) THEN
			nState := 10;
		END_IF

	5:
		bBusy := TRUE;
		IF fbMlSvr.Deconfigure(nTimeout := nConfigureTimeout) THEN
			nErrorCode := fbMlSvr.nErrorCode;
			bError := fbMlSvr.bError OR (nErrorCode <> 0);
			bConfigured := FALSE;
			bBusy := FALSE;
			bResetDone := NOT(bError);
			IF bError THEN
				nState := 90;
			ELSIF bReset THEN
				nState := 0;
			ELSE
				nState := 10;
			END_IF
		END_IF

	10:
		bBusy := TRUE;
		fbMlSvr.stPredictionParameter.sMlModelFilePath := sModelJsonFilePath;
		fbMlSvr.stPredictionParameter.sMlSvrNetId := sMlSvrNetId;
		fbMlSvr.stPredictionParameter.eExecutionProvider := eExecutionProvider;
		IF fbMlSvr.Configure(nTimeout := nConfigureTimeout, nPriority := nPriority) THEN
			nErrorCode := fbMlSvr.nErrorCode;
			bError := fbMlSvr.bError OR (nErrorCode <> 0);
			bConfigured := fbMlSvr.bConfigured AND NOT(bError);
			bBusy := FALSE;
			IF bConfigured THEN
				nState := 20;
			ELSE
				nState := 90;
			END_IF
		END_IF

	20:
		bBusy := FALSE;
		bPredictionPending := FALSE;
		IF bEnable AND bConfigured AND NOT(bError) AND NOT(bReset) THEN
			FOR nSequenceIndex := 0 TO 32 DO
				stModelInput.in_input_tensor[0,nSequenceIndex,0] := fTheta + (INT_TO_REAL(nSequenceIndex) * fThetaStep);
				stModelInput.in_input_tensor[0,nSequenceIndex,1] := fThetaDot;
				stModelInput.in_input_tensor[0,nSequenceIndex,2] := fTorque;
				stModelInput.in_input_tensor[0,nSequenceIndex,3] := fTemperature;
			END_FOR
			bPredictionReady := FALSE;
			bPredictionPending := TRUE;
			nState := 30;
		END_IF

	30:
		bBusy := TRUE;
		bPredictionPending := TRUE;
		IF fbMlSvr.Predict(
			pDataIn := ADR(stModelInput),
			nDataInSize := SIZEOF(ST_Wave51HarmonicPriorSmoothL1StructuredInput),
			pDataOut := ADR(stModelOutput),
			nDataOutSize := SIZEOF(ST_Wave51HarmonicPriorSmoothL1StructuredOutput),
			nTimeout := nPredictTimeout,
			nPriority := nPriority) THEN
			nErrorCode := fbMlSvr.nErrorCode;
			bError := fbMlSvr.bError OR (nErrorCode <> 0);
			nMaxInferenceDuration := fbMlSvr.nMaxInferenceDuration;
			bPredictionPending := FALSE;
			bBusy := FALSE;
			IF NOT(bError) THEN
				aPredictionOutput[0] := stModelOutput.out_prediction_tensor[0,0];
				FOR nOutputIndex := 1 TO 8 DO
					aPredictionOutput[nOutputIndex] := 0.0;
				END_FOR
				bPredictionReady := TRUE;
				nState := 20;
			ELSE
				nState := 90;
			END_IF
		END_IF

	90:
		bBusy := FALSE;
		bPredictionPending := FALSE;
		bError := TRUE;
END_CASE

nErrorCode := fbMlSvr.nErrorCode;
nMaxInferenceDuration := fbMlSvr.nMaxInferenceDuration;

END_FUNCTION_BLOCK
